(* CODESYS project XBoxControllerUtilities.library
   Author: John Helfrich
   Placeholder: XBoxControllerUtilities
   Title: XBoxControllerUtilities
   Version: 1.0
   Company: Beckhoff Community

Project tree, tasks and I/O mapping:
  libraries: Tc2_MC2, * (Beckhoff Automation GmbH); Tc2_Standard, * (Beckhoff Automation GmbH); Tc2_System, * (Beckhoff Automation GmbH); Tc3_Module, * (Beckhoff Automation GmbH)
  DUTs/
    LowerLevel/
      data type ST_XBox_Controller_Buttons_Bits
      data type ST_XBox_Controller_State_Bits2
    XBox NC/
      data type ST_XBox_Button_NC_Options
      data type ST_XBox_Dual_Directional_Joystick_NC_Options
      data type ST_XBox_Single_Directional_Joystick_NC_Options
      data type ST_XBox_Trigger_NC_Options
    data type E_XBox_Controller_Battery_Levels
    data type E_XBox_Controller_Battery_Types
    data type ST_XBox_Class_Command_Status
    data type ST_XBox_Controller_ADS_Inputs
    data type ST_XBox_Controller_Buttons
    data type ST_XBox_Controller_DPad
    data type ST_XBox_Controller_Joystick
    data type ST_XBox_Controller_Rumble
    data type ST_XBox_Controller_Status
  FBs/
    Base Gamepad/
      function block FB_XBox_Controller [ST]: Cycle, FB_init, P_Buttons, P_Left_Joystick, P_Left_Trigger, P_Right_Joystick, P_Right_Trigger, P_SetRumble, P_Status, SetRumble
    NC/
      Buttons/
        function block FB_XBox_Dual_Button_NC [ST]: FB_init, Jog
        function block FB_XBox_Single_Button_NC [ST]: FB_init, Jog
      Joysticks/
        function block FB_XBox_Dual_Directional_Joystick_NC [ST]: FB_init, Jog
        function block FB_XBox_Single_Directional_Joystick_NC [ST]: FB_init, Jog
      Triggers/
        function block FB_XBox_Dual_Trigger_NC [ST]: FB_init, Jog
        function block FB_XBox_Single_Trigger_NC [ST]: FB_init, Jog
  Project Information/
    function F_GetCompany [ST]
    function F_GetTitle [ST]
    function F_GetVersion [ST]
  Version/
    global variables Global_Version
*)

// DUTs/LowerLevel/ST_XBox_Controller_Buttons_Bits
TYPE ST_XBox_Controller_Buttons_Bits :
STRUCT
	xDPAD_UP  			: BIT;
    xDPAD_DOWN  		: BIT;
    xDPAD_LEFT  		: BIT;
    xDPAD_RIGHT  		: BIT;
    xSTART  			: BIT;
    xBACK  				: BIT;
    xLEFT_THUMB  		: BIT;
    xRIGHT_THUMB  		: BIT;   
	xLEFT_SHOULDER  	: BIT;
    xRIGHT_SHOULDER  	: BIT;
	{attribute 'hide'}
	xFiller1 			: BIT;
	{attribute 'hide'}
	xFiller2			: BIT;
	xA  				: BIT;
	xB  				: BIT;
	xX  				: BIT;
	xY  				: BIT;
END_STRUCT
END_TYPE

// DUTs/LowerLevel/ST_XBox_Controller_State_Bits2
TYPE ST_XBox_Controller_State_Bits2 :
STRUCT
	xConnected  				: BIT;
	xBattery_Type_Disconnected	: BIT;
	xBattery_Type_Wired			: BIT;
	xBattery_Type_Alkaline		: BIT;
	xBattery_Type_NIMH			: BIT;
	xBattery_Type_Unknown		: BIT;
	xBattery_Level_Empty		: BIT;
	xBattery_Level_Low			: BIT;
	xBattery_Level_Medium		: BIT;
	xBattery_Level_Full			: BIT;
	
	{attribute 'hide'}
	xFiller10					: BIT;
	{attribute 'hide'}
	xFiller11					: BIT;
	{attribute 'hide'}
	xFiller12					: BIT;
	{attribute 'hide'}
	xFiller13					: BIT;
	{attribute 'hide'}
	xFiller14					: BIT;
	{attribute 'hide'}
	xFiller15					: BIT;
END_STRUCT
END_TYPE

// DUTs/XBox NC/ST_XBox_Button_NC_Options
TYPE ST_XBox_Button_NC_Options :
STRUCT
	// Inverts the direction of the axis
	bInverted : BOOL := FALSE;
	// Maximum Feedrate
	fMaxOverride : LREAL := 100.0;
	// Ramped Feedrate - Increase the feedrate over time of button pressed
	bRampedOverride : BOOL := TRUE;
	// Ramp Step - How often to increase override as button is pressed
	tRampStepTime : TIME := T#100MS;
	// Ramp Step Factor - The % override to step at each time period
	iRampStepFactor : INT := 5;
END_STRUCT
END_TYPE

// DUTs/XBox NC/ST_XBox_Dual_Directional_Joystick_NC_Options
TYPE ST_XBox_Dual_Directional_Joystick_NC_Options :
STRUCT
	// Inverts the direction of the X axis
	bInverted_X : BOOL := FALSE;
	// Inverts the direction of the Y axis
	bInverted_Y : BOOL := FALSE;
	// Maximum Feedrate X Axis
	fMaxOverride_X : LREAL := 100.0;
	// Maximum Feedrate Y Axis
	fMaxOverride_Y : LREAL := 100.0;
END_STRUCT
END_TYPE

// DUTs/XBox NC/ST_XBox_Single_Directional_Joystick_NC_Options
TYPE ST_XBox_Single_Directional_Joystick_NC_Options :
STRUCT
	// Inverts the direction of the axis
	bInverted : BOOL := FALSE;
	// Maximum Feedrate
	fMaxOverride : LREAL := 100.0;
END_STRUCT
END_TYPE

// DUTs/XBox NC/ST_XBox_Trigger_NC_Options
TYPE ST_XBox_Trigger_NC_Options :
STRUCT
	// Inverts the direction of the axis
	bInverted : BOOL := FALSE;
	// Maximum Feedrate
	fMaxOverride : LREAL := 100.0;
END_STRUCT
END_TYPE

// DUTs/E_XBox_Controller_Battery_Levels
{attribute 'qualified_only'}
{attribute 'strict'}
TYPE E_XBox_Controller_Battery_Levels :
(
	// Battery is Empty or Unknown
	Empty := 0,
	// Battery is at low level
	Low := 1,
	// Battery is at medium level
	Medium := 2,
	// Battery is at full level
	Full := 3
);
END_TYPE

// DUTs/E_XBox_Controller_Battery_Types
{attribute 'qualified_only'}
{attribute 'strict'}
TYPE E_XBox_Controller_Battery_Types :
(
	// Battery is disconnected
	Disconnected := 0,
	// Battery is wired
	Wired := 1,
	// Battery is alkaline
	Alkaline := 2,
	// Battery is nickel-metal hydride
	NIMH := 3,
	// Battery is unknown
	Unknown := 4
);
END_TYPE

// DUTs/ST_XBox_Class_Command_Status
TYPE ST_XBox_Class_Command_Status :
STRUCT
	// Command has been completed
	bDone 	: BOOL;
	// Command is busy
	bBusy 	: BOOL;
	// Command has an error
	bError 	: BOOL;
END_STRUCT
END_TYPE

// DUTs/ST_XBox_Controller_ADS_Inputs
TYPE ST_XBox_Controller_ADS_Inputs :
STRUCT
	// Controller Number
	iControllerNumber	: INT;
	// Struct of Left Joystick values
	stLeft_Joystick 	: ST_XBox_Controller_Joystick;
	// Struct of Right Joystick values
	stRight_Joystick 	: ST_XBox_Controller_Joystick;
	// Left Trigger value
	fLeft_Trigger 		: REAL;
	// Right Trigger value
	fRight_Trigger 		: REAL;
	// Struct of individual raw button bits read from the controller
	bButtons 			: ST_XBox_Controller_Buttons_Bits;
	// Struct of individual raw status bits read from the controller
	bStatus				: ST_XBox_Controller_State_Bits2;
END_STRUCT
END_TYPE

// DUTs/ST_XBox_Controller_Buttons
TYPE ST_XBox_Controller_Buttons :
STRUCT
	// Directional Pad Struct
	DPad				: ST_XBox_Controller_DPad;
	// Start Button
    bStart  			: BOOL;
	// Back Button
    bBack  				: BOOL;
	// Pressing in the Left Thumbstick
    bLeft_Thumbstick  	: BOOL;
	// Pressing in the Right Thumbstick
    bRight_Thumbstick  	: BOOL;
	// Left Shoulder Button  
	bLeft_Shoulder  	: BOOL;
	// Right Shoulder Button
    bRight_Shoulder  	: BOOL;
	// Button A
	bA_Button  			: BOOL;
	// Button B
	bB_Button  			: BOOL;
	// Button X
	bX_Button  			: BOOL;
	// Button Y
	bY_Button  			: BOOL;
END_STRUCT
END_TYPE

// DUTs/ST_XBox_Controller_DPad
TYPE ST_XBox_Controller_DPad :
STRUCT
	// Up Button on DPad
	bUp  		: BOOL;
	// Down Button on DPad
    bDown  		: BOOL;
	// Left Button on DPad
    bLeft  		: BOOL;
	// Right Button on DPad
    bRight  	: BOOL;
END_STRUCT
END_TYPE

// DUTs/ST_XBox_Controller_Joystick
TYPE ST_XBox_Controller_Joystick :
STRUCT
	// Joystick's X Value (-100...100%)
	fX : REAL;
	// Joystick's Y Value (-100...100%)
	fY : REAL;
END_STRUCT
END_TYPE

// DUTs/ST_XBox_Controller_Rumble
TYPE ST_XBox_Controller_Rumble :
STRUCT
	// Rumble of left motor (0..100%)
	fLeftMotor 	: REAL;
	// Rumble of right motor (0..100%)
	fRightMotor : REAL;
END_STRUCT
END_TYPE

// DUTs/ST_XBox_Controller_Status
TYPE ST_XBox_Controller_Status :
STRUCT
	// Controller's ID
	iControllerNumber  	: INT;
	// Controller is connected to the PC
	bConnected  		: BOOL;
	// Controller is disconnected from the PC
	bDisconnected  		: BOOL;
	// Battery Type
	Battery_Type 		: E_XBox_Controller_Battery_Types;
	// Battery Level
	Battery_Level 		: E_XBox_Controller_Battery_Levels;
END_STRUCT
END_TYPE

// Version/Global_Version
{attribute 'TcGenerated'}
{attribute 'no-analysis'}
{attribute 'linkalways'}
// This function has been automatically generated from the project information.
VAR_GLOBAL CONSTANT
	{attribute 'const_non_replaced'}
	stLibVersion_XBoxControllerUtilities : ST_LibVersion := (iMajor := 1, iMinor := 0, iBuild := 0, iRevision := 0, nFlags := 1, sVersion := '1.0');
END_VAR

// FBs/Base Gamepad/FB_XBox_Controller
FUNCTION_BLOCK FB_XBox_Controller
VAR
	{attribute 'hide'}
	_AmsNetId : T_AMSNETID;
	{attribute 'hide'}
	_WriteServerData : ADSWRITE;
	{attribute 'hide'}
	_ReadServerData : ADSREAD;
	// RAW ADS Inputs for debug (Use properties to access items)
	stXBoxControllerInputs : ST_XBox_Controller_ADS_Inputs;
	{attribute 'hide'}
	_stRumble : ST_XBox_Controller_Rumble;
	{attribute 'hide'}
	_IDXGRP : UDINT;
	{attribute 'hide'}
	_rumbleCommand 			: ST_XBox_Class_Command_Status;
	{attribute 'hide'}
	_stControllerButtons 	: ST_XBox_Controller_Buttons;
	{attribute 'hide'}
	_stControllerStatus		: ST_XBox_Controller_Status;
	{attribute 'hide'}
	_stLeftJoystick 		: ST_XBox_Controller_Joystick;
	{attribute 'hide'}
	_stRightJoystick 		: ST_XBox_Controller_Joystick;
	{attribute 'hide'}
	_fLeftTrigger 			: REAL;
	{attribute 'hide'}
	_fRightTrigger 			: REAL;
	{attribute 'hide'}
	_bSetRumbleEvent 		: BOOL; // Internal indication of an ADS write event
	{attribute 'hide'}
	_bSetRumbleEventLogged	: BOOL; // Check if the Set Rumble event is being called too many times	
END_VAR

// This method is called cyclically to update the controller inputs
METHOD Cycle : BOOL
// Read the current inputs
THIS^._ReadServerData(
	NETID:= THIS^._AmsNetId, 
	PORT:= 25733, 
	IDXGRP:= THIS^._IDXGRP, 
	IDXOFFS:= 0, 
	LEN:= SIZEOF(THIS^.stXBoxControllerInputs), 
	DESTADDR:= ADR(THIS^.stXBoxControllerInputs), 
	READ:= TRUE, 
	TMOUT:= T#5S,
	ERR=>);
	
// If there is an error in reading from the server, shut all inputs off
IF THIS^._ReadServerData.ERR THEN
	memset(ADR(THIS^.stXBoxControllerInputs), 0, SIZEOF(THIS^.stXBoxControllerInputs));
END_IF

// Stop read command
THIS^._ReadServerData(
	NETID:= THIS^._AmsNetId, 
	PORT:= 25733, 
	IDXGRP:= THIS^._IDXGRP, 
	IDXOFFS:= 0, 
	LEN:= SIZEOF(THIS^.stXBoxControllerInputs), 
	DESTADDR:= ADR(THIS^.stXBoxControllerInputs), 
	READ:= FALSE, 
	TMOUT:= T#5S,
	ERR=>);
	

// Handle any write requests for the rumble
// Write the new values
THIS^._WriteServerData(
	NETID:= THIS^._AmsNetId, 
	PORT:= 25733, 
	IDXGRP:= THIS^._IDXGRP, 
	IDXOFFS:= 16, 
	LEN:= SIZEOF(THIS^._stRumble), 
	SRCADDR:= ADR(THIS^._stRumble), 
	WRITE:= THIS^._bSetRumbleEvent, 
	TMOUT:= T#5S);
	
// Update the status of the current command if active
IF 	THIS^._bSetRumbleEvent THEN
	THIS^.P_SetRumble.bBusy := THIS^._WriteServerData.BUSY;
	THIS^.P_SetRumble.bError := THIS^._WriteServerData.ERR;
END_IF

// Check if it's done writing
IF THIS^._bSetRumbleEvent AND NOT THIS^._WriteServerData.BUSY THEN
	IF NOT THIS^._WriteServerData.ERR THEN
		THIS^.P_SetRumble.bDone := TRUE;
	END_IF
	// Turn off the write request
	THIS^._WriteServerData(
		NETID:= THIS^._AmsNetId, 
		PORT:= 25733, 
		IDXGRP:= THIS^._IDXGRP, 
		IDXOFFS:= 16, 
		LEN:= SIZEOF(THIS^._stRumble), 
		SRCADDR:= ADR(THIS^._stRumble), 
		WRITE:= FALSE, 
		TMOUT:= T#5S);
		
	THIS^._bSetRumbleEvent := FALSE;
END_IF
END_METHOD

METHOD FB_init : BOOL
VAR_INPUT
	bInitRetains : BOOL; // if TRUE, the retain variables are initialized (warm start / cold start)
	bInCopyCode : BOOL;  // if TRUE, the instance afterwards gets moved into the copy code (online change)
	NetID 				: T_AMSNETID := ''; // AMS Net ID of the XBox Service Provider
	iControllerNumber 	: UINT(1..4) := 1; // The controller number for the controller you'd like to use
END_VAR
THIS^._AmsNetId := NetID;
THIS^._IDXGRP := iControllerNumber * 16#10000;
END_METHOD

// Structure of the different active buttons
PROPERTY P_Buttons : REFERENCE TO ST_XBox_Controller_Buttons
GET
IF THIS^.stXBoxControllerInputs.bStatus.xConnected THEN	
	THIS^._stControllerButtons.DPad.bUp				:= THIS^.stXBoxControllerInputs.bButtons.xDPAD_UP;
	THIS^._stControllerButtons.DPad.bDown			:= THIS^.stXBoxControllerInputs.bButtons.xDPAD_DOWN;
	THIS^._stControllerButtons.DPad.bLeft			:= THIS^.stXBoxControllerInputs.bButtons.xDPAD_LEFT;
	THIS^._stControllerButtons.DPad.bRight			:= THIS^.stXBoxControllerInputs.bButtons.xDPAD_RIGHT;
	THIS^._stControllerButtons.bStart  				:= THIS^.stXBoxControllerInputs.bButtons.xSTART;
	THIS^._stControllerButtons.bBack  				:= THIS^.stXBoxControllerInputs.bButtons.xBACK;
	THIS^._stControllerButtons.bLeft_Thumbstick  	:= THIS^.stXBoxControllerInputs.bButtons.xLEFT_THUMB;
	THIS^._stControllerButtons.bRight_Thumbstick 	:= THIS^.stXBoxControllerInputs.bButtons.xRIGHT_THUMB;
	THIS^._stControllerButtons.bLeft_Shoulder  		:= THIS^.stXBoxControllerInputs.bButtons.xLEFT_SHOULDER;
	THIS^._stControllerButtons.bRight_Shoulder  	:= THIS^.stXBoxControllerInputs.bButtons.xRIGHT_SHOULDER;
	THIS^._stControllerButtons.bA_Button  			:= THIS^.stXBoxControllerInputs.bButtons.xA;
	THIS^._stControllerButtons.bB_Button  			:= THIS^.stXBoxControllerInputs.bButtons.xB;
	THIS^._stControllerButtons.bX_Button  			:= THIS^.stXBoxControllerInputs.bButtons.xX;
	THIS^._stControllerButtons.bY_Button  			:= THIS^.stXBoxControllerInputs.bButtons.xY;
ELSE
	THIS^._stControllerButtons.DPad.bUp				:= FALSE;
	THIS^._stControllerButtons.DPad.bDown			:= FALSE;
	THIS^._stControllerButtons.DPad.bLeft			:= FALSE;
	THIS^._stControllerButtons.DPad.bRight			:= FALSE;
	THIS^._stControllerButtons.bStart  				:= FALSE;
	THIS^._stControllerButtons.bBack  				:= FALSE;
	THIS^._stControllerButtons.bLeft_Thumbstick  	:= FALSE;
	THIS^._stControllerButtons.bRight_Thumbstick 	:= FALSE;
	THIS^._stControllerButtons.bLeft_Shoulder  		:= FALSE;
	THIS^._stControllerButtons.bRight_Shoulder  	:= FALSE;
	THIS^._stControllerButtons.bA_Button  			:= FALSE;
	THIS^._stControllerButtons.bB_Button  			:= FALSE;
	THIS^._stControllerButtons.bX_Button  			:= FALSE;
	THIS^._stControllerButtons.bY_Button  			:= FALSE;
END_IF
P_Buttons REF= THIS^._stControllerButtons;
END_GET
END_PROPERTY

// Returns a structure of data for the XY Joystick values
PROPERTY P_Left_Joystick : REFERENCE TO ST_XBox_Controller_Joystick
GET
IF THIS^.stXBoxControllerInputs.bStatus.xConnected THEN	
	THIS^._stLeftJoystick.fX := THIS^.stXBoxControllerInputs.stLeft_Joystick.fX;
	THIS^._stLeftJoystick.fY := THIS^.stXBoxControllerInputs.stLeft_Joystick.fY;
ELSE
	THIS^._stLeftJoystick.fX := 0;
	THIS^._stLeftJoystick.fY := 0;
END_IF
P_Left_Joystick REF= THIS^._stLeftJoystick;
END_GET
END_PROPERTY

// Left trigger value
PROPERTY P_Left_Trigger : REFERENCE TO REAL
GET
IF THIS^.stXBoxControllerInputs.bStatus.xConnected THEN	
	THIS^._fLeftTrigger := THIS^.stXBoxControllerInputs.fLeft_Trigger;
ELSE
	THIS^._fLeftTrigger := 0;
END_IF
P_Left_Trigger REF= THIS^._fLeftTrigger;
END_GET
END_PROPERTY

// Returns a structure of data for the XY Joystick values
PROPERTY P_Right_Joystick : REFERENCE TO ST_XBox_Controller_Joystick
GET
IF THIS^.stXBoxControllerInputs.bStatus.xConnected THEN	
	THIS^._stRightJoystick.fX := THIS^.stXBoxControllerInputs.stRight_Joystick.fX;
	THIS^._stRightJoystick.fY := THIS^.stXBoxControllerInputs.stRight_Joystick.fY;
ELSE
	THIS^._stRightJoystick.fX := 0;
	THIS^._stRightJoystick.fY := 0;
END_IF
P_Right_Joystick REF= THIS^._stRightJoystick;
END_GET
END_PROPERTY

// Right trigger value
PROPERTY P_Right_Trigger : REFERENCE TO REAL
GET
IF THIS^.stXBoxControllerInputs.bStatus.xConnected THEN	
	THIS^._fRightTrigger := THIS^.stXBoxControllerInputs.fRight_Trigger;
ELSE
	THIS^._fRightTrigger := 0;
END_IF
P_Right_Trigger REF= THIS^._fRightTrigger;
END_GET
END_PROPERTY

// Status of the SetRumble method
PROPERTY P_SetRumble : REFERENCE TO ST_XBox_Class_Command_Status
GET
P_SetRumble REF= THIS^._rumbleCommand;
END_GET
END_PROPERTY

// Structure of the controller capabilites and status
PROPERTY P_Status : REFERENCE TO ST_XBox_Controller_Status
GET
IF THIS^.stXBoxControllerInputs.bStatus.xConnected THEN	
	THIS^._stControllerStatus.bConnected 		:= TRUE;
	THIS^._stControllerStatus.bDisconnected 	:= FALSE;
	THIS^._stControllerStatus.iControllerNumber := THIS^.stXBoxControllerInputs.iControllerNumber;
ELSE
	THIS^._stControllerStatus.bConnected 		:= FALSE;
	THIS^._stControllerStatus.bDisconnected 	:= TRUE;
	THIS^._stControllerStatus.iControllerNumber := 0;
END_IF

IF THIS^.stXBoxControllerInputs.bStatus.xBattery_Type_Disconnected THEN
	THIS^._stControllerStatus.Battery_Type := E_XBox_Controller_Battery_Types.Disconnected;
END_IF

IF THIS^.stXBoxControllerInputs.bStatus.xBattery_Type_Wired THEN
	THIS^._stControllerStatus.Battery_Type := E_XBox_Controller_Battery_Types.Wired;
END_IF

IF THIS^.stXBoxControllerInputs.bStatus.xBattery_Type_Alkaline THEN
	THIS^._stControllerStatus.Battery_Type := E_XBox_Controller_Battery_Types.Alkaline;
END_IF

IF THIS^.stXBoxControllerInputs.bStatus.xBattery_Type_NIMH THEN
	THIS^._stControllerStatus.Battery_Type := E_XBox_Controller_Battery_Types.NIMH;
END_IF

IF THIS^.stXBoxControllerInputs.bStatus.xBattery_Type_Unknown THEN
	THIS^._stControllerStatus.Battery_Type := E_XBox_Controller_Battery_Types.Unknown;
END_IF

IF THIS^.stXBoxControllerInputs.bStatus.xBattery_Level_Empty THEN
	THIS^._stControllerStatus.Battery_Level := E_XBox_Controller_Battery_Levels.Empty;
END_IF

IF THIS^.stXBoxControllerInputs.bStatus.xBattery_Level_Low THEN
	THIS^._stControllerStatus.Battery_Level := E_XBox_Controller_Battery_Levels.Low;
END_IF

IF THIS^.stXBoxControllerInputs.bStatus.xBattery_Level_Medium THEN
	THIS^._stControllerStatus.Battery_Level := E_XBox_Controller_Battery_Levels.Medium;
END_IF

IF THIS^.stXBoxControllerInputs.bStatus.xBattery_Level_Full THEN
	THIS^._stControllerStatus.Battery_Level := E_XBox_Controller_Battery_Levels.Full;
END_IF


P_Status REF= THIS^._stControllerStatus;
END_GET
END_PROPERTY

// Sets the rumble for the controller
METHOD SetRumble : BOOL
VAR_INPUT
	// Left motor speed (0..100%)
	fLeftMotor : REAL;
	// Right motor speed (0..100%)
	fRightMotor : REAL;
END_VAR
// When the method is called, check if a write is in progress
IF THIS^._bSetRumbleEvent THEN
	// ADS you are doing that too much
	IF NOT THIS^._bSetRumbleEventLogged THEN
		ADSLOGSTR( msgCtrlMask := ADSLOG_MSGTYPE_WARN, msgFmtStr := 'PLC Msg.: Command being called too often, wait for done bit: %s', strArg := 'SetRumble()');
		THIS^._bSetRumbleEventLogged := TRUE;
	END_IF	
ELSE
	// Check if the value is within range
	IF fLeftMotor > 100 THEN
		THIS^._stRumble.fLeftMotor := 100.0;
	ELSIF fLeftMotor < 0 THEN
		THIS^._stRumble.fLeftMotor := 0.0;
	ELSE
		THIS^._stRumble.fLeftMotor := fLeftMotor;
	END_IF
	
	// Check if the value is within range
	IF fRightMotor > 100 THEN
		THIS^._stRumble.fRightMotor := 100.0;
	ELSIF fRightMotor < 0 THEN
		THIS^._stRumble.fRightMotor := 0.0;
	ELSE
		THIS^._stRumble.fRightMotor := fRightMotor;
	END_IF
	
	//Reset all status for the command
	THIS^.P_SetRumble.bDone := FALSE;
	THIS^.P_SetRumble.bBusy := FALSE;
	THIS^.P_SetRumble.bError := FALSE;

	// Set the high bit on the write command
	THIS^._bSetRumbleEvent := TRUE;
END_IF

// If it's done, set the current even in progress to false
IF P_SetRumble.bDone THEN
	THIS^._bSetRumbleEvent := FALSE;
END_IF

// Event Received
SetRumble := THIS^._bSetRumbleEvent;
END_METHOD

END_FUNCTION_BLOCK

// FBs/NC/Buttons/FB_XBox_Dual_Button_NC
FUNCTION_BLOCK FB_XBox_Dual_Button_NC
VAR
	// Axis Control Blocks
	_Button_NC			: FB_XBox_Single_Button_NC;
	_rtJogEnable		: R_TRIG;
	_ftJogEnable		: F_TRIG;
	_fPrevOverride		: UDINT;
END_VAR

METHOD FB_init : BOOL
VAR_INPUT
	bInitRetains : BOOL; // if TRUE, the retain variables are initialized (warm start / cold start)
	bInCopyCode : BOOL;  // if TRUE, the instance afterwards gets moved into the copy code (online change)
END_VAR
END_METHOD

METHOD Jog : BOOL
VAR_INPUT
	bEnable				: BOOL;	
	bForward_Button		: BOOL;
	bBackwards_Button	: BOOL;
	Axis				: REFERENCE TO Axis_Ref;
	stOptions			: ST_XBox_Button_NC_Options;
END_VAR
VAR	
	stButtonOptions		: ST_XBox_Button_NC_Options;
	bButtonCommand		: BOOL;
END_VAR
// Rising edge trigger of the block enable
_rtJogEnable(CLK := bEnable);
// Falling edge trigger of the block enable
_ftJogEnable(CLK := bEnable);

IF __ISVALIDREF(Axis) THEN
	// Rising edge trigger of the block enable
	IF _rtJogEnable.Q THEN
		// Save the current override value before jogging
		THIS^._fPrevOverride := Axis.PlcToNc.Override;
	END_IF
	
	// Figure out what direction the axis should move
	IF bForward_Button AND bBackwards_Button THEN
		bButtonCommand := FALSE;
	ELSIF bForward_Button THEN
		bButtonCommand := bForward_Button;
		IF NOT stOptions.bInverted THEN
			stButtonOptions.bInverted := FALSE;
		ELSE
			stButtonOptions.bInverted := TRUE;
		END_IF
	ELSIF bBackwards_Button THEN
		bButtonCommand := bBackwards_Button;
		IF NOT stOptions.bInverted THEN
			stButtonOptions.bInverted := TRUE;
		ELSE
			stButtonOptions.bInverted := FALSE;
		END_IF
	ELSE
		bButtonCommand := FALSE;
	END_IF
	
	stButtonOptions.bRampedOverride := stOptions.bRampedOverride;
	stButtonOptions.fMaxOverride := stOptions.fMaxOverride;
	stButtonOptions.iRampStepFactor := stOptions.iRampStepFactor;
	stButtonOptions.tRampStepTime := stOptions.tRampStepTime;
	
	// Jog the axis
	_Button_NC.Jog(bEnable:= bEnable, bButton:= bButtonCommand, Axis:= Axis, stOptions:= stButtonOptions);
	
	// Falling edge trigger of the block enable
	IF _ftJogEnable.Q THEN
		// Restore the past override value before enable
		Axis.PlcToNc.Override := THIS^._fPrevOverride;
	END_IF
END_IF
END_METHOD

END_FUNCTION_BLOCK

// FBs/NC/Buttons/FB_XBox_Single_Button_NC
FUNCTION_BLOCK FB_XBox_Single_Button_NC
VAR
	_mcJog				: MC_Jog;
	_rtJogEnable		: R_TRIG;
	_ftJogEnable		: F_TRIG;
	_bJoggingActive		: BOOL;
	_fPrevOverride		: UDINT;
	_RampTimer			: TON;
	_fCurrentOverride   : LREAL;
END_VAR

METHOD FB_init : BOOL
VAR_INPUT
	bInitRetains : BOOL; // if TRUE, the retain variables are initialized (warm start / cold start)
	bInCopyCode : BOOL;  // if TRUE, the instance afterwards gets moved into the copy code (online change)
END_VAR
END_METHOD

METHOD Jog : BOOL
VAR_INPUT
	bEnable			: BOOL;	
	bButton			: BOOL;
	Axis			: REFERENCE TO Axis_Ref;
	stOptions		: ST_XBox_Button_NC_Options;
END_VAR
VAR
	bJogForward 	 : BOOL;
	bJogBackwards 	 : BOOL;
END_VAR
// Rising edge trigger of the block enable
_rtJogEnable(CLK := bEnable);
// Falling edge trigger of the block enable
_ftJogEnable(CLK := bEnable);

// Rising edge trigger of the block enable
IF _rtJogEnable.Q THEN
	// Save the current override value before jogging
	// Check the Axis reference is valid	
	IF __ISVALIDREF(Axis) THEN
		THIS^._fPrevOverride := Axis.PlcToNc.Override;
	END_IF
	// Enable the jog methods
	_bJoggingActive	:= TRUE;
END_IF

// Falling edge trigger of the block enable
IF _ftJogEnable.Q THEN
	// Restore the past override value before enable
	// Check the Axis reference is valid	
	IF __ISVALIDREF(Axis) THEN
		Axis.PlcToNc.Override := THIS^._fPrevOverride;
			// Cleanup any old Jog commands
		THIS^._mcJog(
					  Axis:= Axis, 
					  JogForward:= FALSE, 
					  JogBackwards:= FALSE, 
					  Mode:= E_JogMode.MC_JOGMODE_STANDARD_FAST);	
	END_IF
	// Disable calling to jog methods
	_bJoggingActive := FALSE;
END_IF

// Check the Joystick reference is valid
IF _bJoggingActive THEN
	// Check the Axis reference is valid	
	IF __ISVALIDREF(Axis) THEN
		// Speed Ramp Timer
		_RampTimer(IN:=stOptions.bRampedOverride AND NOT _RampTimer.Q, PT:= stOptions.tRampStepTime);
		
		// Check the direction the joystick is moving, or if in deadzone					 
		IF bButton = FALSE THEN
			bJogForward 	:= FALSE;
			bJogBackwards := FALSE;
			Axis.PlcToNc.Override := 0;
			_fCurrentOverride := 0;
		ELSE
			// Check for inversion
			IF NOT stOptions.bInverted THEN
				bJogForward 	:= TRUE;
				bJogBackwards 	:= FALSE;
			ELSE
				bJogForward 	:= FALSE;
				bJogBackwards 	:= TRUE;
			END_IF
			
			// Find the override speed

			IF _RampTimer.Q AND stOptions.bRampedOverride THEN
				_fCurrentOverride := _fCurrentOverride + stOptions.iRampStepFactor;		
			ELSIF NOT stOptions.bRampedOverride THEN
				_fCurrentOverride := stOptions.fMaxOverride;
			END_IF
			// Check range
			IF _fCurrentOverride > stOptions.fMaxOverride THEN
				_fCurrentOverride := stOptions.fMaxOverride;
			END_IF
			
			Axis.PlcToNc.Override := TO_UDINT(ABS(_fCurrentOverride) * 10000);
		END_IF
		
		// Main jog call for axis
		THIS^._mcJog(
					  Axis:= Axis, 
					  JogForward:= bJogForward, 
					  JogBackwards:= bJogBackwards, 
					  Mode:= E_JogMode.MC_JOGMODE_STANDARD_FAST);
	END_IF
END_IF
END_METHOD

END_FUNCTION_BLOCK

// FBs/NC/Joysticks/FB_XBox_Dual_Directional_Joystick_NC
FUNCTION_BLOCK FB_XBox_Dual_Directional_Joystick_NC
VAR
	// Axis Control Blocks
	_JoystickNC_X		: FB_XBox_Single_Directional_Joystick_NC;
	_JoystickNC_Y		: FB_XBox_Single_Directional_Joystick_NC;
END_VAR

METHOD FB_init : BOOL
VAR_INPUT
	bInitRetains : BOOL; // if TRUE, the retain variables are initialized (warm start / cold start)
	bInCopyCode : BOOL;  // if TRUE, the instance afterwards gets moved into the copy code (online change)
END_VAR
END_METHOD

METHOD Jog
VAR_INPUT
	bEnable			: BOOL;	
	stJoystick		: REFERENCE TO ST_XBox_Controller_Joystick;
	X_Axis			: REFERENCE TO Axis_Ref;
	Y_Axis			: REFERENCE TO Axis_Ref;
	stOptions		: ST_XBox_Dual_Directional_Joystick_NC_Options;
END_VAR
VAR	
	X_Axis_Options: ST_XBox_Single_Directional_Joystick_NC_Options;
	Y_Axis_Options: ST_XBox_Single_Directional_Joystick_NC_Options;
END_VAR
IF __ISVALIDREF(stJoystick) AND __ISVALIDREF(X_Axis) AND __ISVALIDREF(Y_Axis) THEN
	// Call the X-Axis Joystick
	X_Axis_Options.bInverted := stOptions.bInverted_X;
	X_Axis_Options.fMaxOverride := stOptions.fMaxOverride_X;
	_JoystickNC_X.Jog(bEnable:= bEnable, fJoystick:= stJoystick.fX, Axis:= X_Axis, stOptions:= X_Axis_Options);
	
	// Call the Y-Axis Joystick
	Y_Axis_Options.bInverted := stOptions.bInverted_Y;
	Y_Axis_Options.fMaxOverride := stOptions.fMaxOverride_Y;
	_JoystickNC_Y.Jog(bEnable:= bEnable, fJoystick:= stJoystick.fY, Axis:= Y_Axis, stOptions:= Y_Axis_Options);
END_IF
END_METHOD

END_FUNCTION_BLOCK

// FBs/NC/Joysticks/FB_XBox_Single_Directional_Joystick_NC
FUNCTION_BLOCK FB_XBox_Single_Directional_Joystick_NC
VAR
	_mcJog				: MC_Jog;
	_rtJogEnable		: R_TRIG;
	_ftJogEnable		: F_TRIG;
	_bJoggingActive		: BOOL;
	_fPrevOverride		: UDINT;
END_VAR

METHOD FB_init : BOOL
VAR_INPUT
	bInitRetains : BOOL; // if TRUE, the retain variables are initialized (warm start / cold start)
	bInCopyCode : BOOL;  // if TRUE, the instance afterwards gets moved into the copy code (online change)
END_VAR
END_METHOD

METHOD Jog
VAR_INPUT
	bEnable			: BOOL;	
	fJoystick		: LREAL;
	Axis			: REFERENCE TO Axis_Ref;
	stOptions		: ST_XBox_Single_Directional_Joystick_NC_Options;
END_VAR
VAR
	bJogForward 	: BOOL;
	bJogBackwards 	: BOOL;
END_VAR
// Rising edge trigger of the block enable
_rtJogEnable(CLK := bEnable);
// Falling edge trigger of the block enable
_ftJogEnable(CLK := bEnable);

// Rising edge trigger of the block enable
IF _rtJogEnable.Q THEN
	// Save the current override value before jogging
	// Check the Axis reference is valid	
	IF __ISVALIDREF(Axis) THEN
		THIS^._fPrevOverride := Axis.PlcToNc.Override;
	END_IF
	// Enable the jog methods
	_bJoggingActive	:= TRUE;
END_IF

// Falling edge trigger of the block enable
IF _ftJogEnable.Q THEN
	// Restore the past override value before enable
	// Check the Axis reference is valid	
	IF __ISVALIDREF(Axis) THEN
		Axis.PlcToNc.Override := THIS^._fPrevOverride;
			// Cleanup any old Jog commands
		THIS^._mcJog(
					  Axis:= Axis, 
					  JogForward:= FALSE, 
					  JogBackwards:= FALSE, 
					  Mode:= E_JogMode.MC_JOGMODE_STANDARD_FAST);	
	END_IF
	// Disable calling to jog methods
	_bJoggingActive := FALSE;
END_IF

// Check the Joystick reference is valid
IF _bJoggingActive THEN
	// Check the Axis reference is valid	
	IF __ISVALIDREF(Axis) THEN
		// Check the direction the joystick is moving, or if in deadzone					 
		IF fJoystick = 0 THEN
			bJogForward 	:= FALSE;
			bJogBackwards := FALSE;
			Axis.PlcToNc.Override := 0;
		ELSIF fJoystick < 0 THEN
			// Check for inversion
			IF NOT stOptions.bInverted THEN
				bJogForward 	:= FALSE;
				bJogBackwards := TRUE;
			ELSE
				bJogForward 	:= TRUE;
				bJogBackwards := FALSE;
			END_IF
			// Set the new override based on the directional pressure
			Axis.PlcToNc.Override := TO_UDINT(ABS(fJoystick * (stOptions.fMaxOverride/100)) * 10000);
		ELSIF fJoystick > 0 THEN
			// Check for inversion
			IF NOT stOptions.bInverted THEN
				bJogForward 	:= TRUE;
				bJogBackwards := FALSE;
			ELSE
				bJogForward 	:= FALSE;
				bJogBackwards := TRUE;
			END_IF
			// Set the new override based on the directional pressure
			Axis.PlcToNc.Override := TO_UDINT(ABS(fJoystick * (stOptions.fMaxOverride/100)) * 10000);
		END_IF
		// Main jog call for axis
		THIS^._mcJog(
					  Axis:= Axis, 
					  JogForward:= bJogForward, 
					  JogBackwards:= bJogBackwards, 
					  Mode:= E_JogMode.MC_JOGMODE_STANDARD_FAST);
	END_IF
END_IF
END_METHOD

END_FUNCTION_BLOCK

// FBs/NC/Triggers/FB_XBox_Dual_Trigger_NC
FUNCTION_BLOCK FB_XBox_Dual_Trigger_NC
VAR
	// Axis Control Blocks
	_Trigger_NC			: FB_XBox_Single_Trigger_NC;
	_rtJogEnable		: R_TRIG;
	_ftJogEnable		: F_TRIG;
	_fPrevOverride		: UDINT;
END_VAR

METHOD FB_init : BOOL
VAR_INPUT
	bInitRetains : BOOL; // if TRUE, the retain variables are initialized (warm start / cold start)
	bInCopyCode : BOOL;  // if TRUE, the instance afterwards gets moved into the copy code (online change)
END_VAR
END_METHOD

METHOD Jog
VAR_INPUT
	bEnable			: BOOL;	
	fLeft_Trigger	: LREAL;
	fRight_Trigger	: LREAL;
	Axis			: REFERENCE TO Axis_Ref;
	stOptions		: ST_XBox_Trigger_NC_Options;
END_VAR
VAR	
	stTrigOptions		: ST_XBox_Trigger_NC_Options;
	fTriggerCommand		: LREAL;
END_VAR
// Rising edge trigger of the block enable
_rtJogEnable(CLK := bEnable);
// Falling edge trigger of the block enable
_ftJogEnable(CLK := bEnable);

IF __ISVALIDREF(Axis) THEN
	// Rising edge trigger of the block enable
	IF _rtJogEnable.Q THEN
		// Save the current override value before jogging
		THIS^._fPrevOverride := Axis.PlcToNc.Override;
	END_IF
	
	// Figure out what direction the axis should move
	IF fLeft_Trigger > fRight_Trigger THEN
		fTriggerCommand := fLeft_Trigger;
		IF NOT stOptions.bInverted THEN
			stTrigOptions.bInverted := FALSE;
		ELSE
			stTrigOptions.bInverted := TRUE;
		END_IF
	ELSIF fRight_Trigger > fLeft_Trigger THEN
		fTriggerCommand := fRight_Trigger;
		IF NOT stOptions.bInverted THEN
			stTrigOptions.bInverted := TRUE;
		ELSE
			stTrigOptions.bInverted := FALSE;
		END_IF
	ELSE
		fTriggerCommand := 0;
	END_IF
	stTrigOptions.fMaxOverride := stOptions.fMaxOverride;
	// Jog the axis
	_Trigger_NC.Jog(bEnable:= bEnable, fTrigger:= fTriggerCommand, Axis:= Axis, stOptions:= stTrigOptions);
	
	
	// Falling edge trigger of the block enable
	IF _ftJogEnable.Q THEN
		// Restore the past override value before enable
		Axis.PlcToNc.Override := THIS^._fPrevOverride;
	END_IF
END_IF
END_METHOD

END_FUNCTION_BLOCK

// FBs/NC/Triggers/FB_XBox_Single_Trigger_NC
FUNCTION_BLOCK FB_XBox_Single_Trigger_NC
VAR
	_mcJog				: MC_Jog;
	_rtJogEnable		: R_TRIG;
	_ftJogEnable		: F_TRIG;
	_bJoggingActive		: BOOL;
	_fPrevOverride		: UDINT;
END_VAR

METHOD FB_init : BOOL
VAR_INPUT
	bInitRetains : BOOL; // if TRUE, the retain variables are initialized (warm start / cold start)
	bInCopyCode : BOOL;  // if TRUE, the instance afterwards gets moved into the copy code (online change)
END_VAR
END_METHOD

METHOD Jog
VAR_INPUT
	bEnable			: BOOL;	
	fTrigger		: LREAL;
	Axis			: REFERENCE TO Axis_Ref;
	stOptions		: ST_XBox_Trigger_NC_Options;
END_VAR
VAR
	bJogForward 	: BOOL;
	bJogBackwards 	: BOOL;
END_VAR
// Rising edge trigger of the block enable
_rtJogEnable(CLK := bEnable);
// Falling edge trigger of the block enable
_ftJogEnable(CLK := bEnable);

// Rising edge trigger of the block enable
IF _rtJogEnable.Q THEN
	// Save the current override value before jogging
	// Check the Axis reference is valid	
	IF __ISVALIDREF(Axis) THEN
		THIS^._fPrevOverride := Axis.PlcToNc.Override;
	END_IF
	// Enable the jog methods
	_bJoggingActive	:= TRUE;
END_IF

// Falling edge trigger of the block enable
IF _ftJogEnable.Q THEN
	// Restore the past override value before enable
	// Check the Axis reference is valid	
	IF __ISVALIDREF(Axis) THEN
		Axis.PlcToNc.Override := THIS^._fPrevOverride;
			// Cleanup any old Jog commands
		THIS^._mcJog(
					  Axis:= Axis, 
					  JogForward:= FALSE, 
					  JogBackwards:= FALSE, 
					  Mode:= E_JogMode.MC_JOGMODE_STANDARD_FAST);	
	END_IF
	// Disable calling to jog methods
	_bJoggingActive := FALSE;
END_IF

// Check the Joystick reference is valid
IF _bJoggingActive THEN
	// Check the Axis reference is valid	
	IF __ISVALIDREF(Axis) THEN
		// Check the direction the joystick is moving, or if in deadzone					 
		IF fTrigger = 0 THEN
			bJogForward 	:= FALSE;
			bJogBackwards := FALSE;
			Axis.PlcToNc.Override := 0;
		ELSE
			// Check for inversion
			IF NOT stOptions.bInverted THEN
				bJogForward 	:= TRUE;
				bJogBackwards := FALSE;
			ELSE
				bJogForward 	:= FALSE;
				bJogBackwards := TRUE;
			END_IF
			// Set the new override based on the directional pressure
			Axis.PlcToNc.Override := TO_UDINT(ABS(fTrigger  * (stOptions.fMaxOverride/100)) * 10000);
		END_IF
		
		// Main jog call for axis
		THIS^._mcJog(
					  Axis:= Axis, 
					  JogForward:= bJogForward, 
					  JogBackwards:= bJogBackwards, 
					  Mode:= E_JogMode.MC_JOGMODE_STANDARD_FAST);
	END_IF
END_IF
END_METHOD

END_FUNCTION_BLOCK

// Project Information/F_GetCompany
// This function has been automatically generated from the project information.
{attribute 'signature_flag' := '1073741824'}
{attribute 'TcGenerated'}
{attribute 'no-analysis'}
FUNCTION F_GetCompany : WSTRING
VAR_INPUT
	
END_VAR

F_GetCompany := "Beckhoff Community";

END_FUNCTION

// Project Information/F_GetTitle
// This function has been automatically generated from the project information.
{attribute 'signature_flag' := '1073741824'}
{attribute 'TcGenerated'}
{attribute 'no-analysis'}
FUNCTION F_GetTitle : WSTRING
VAR_INPUT
	
END_VAR

F_GetTitle := "XBoxControllerUtilities";

END_FUNCTION

// Project Information/F_GetVersion
// This function has been automatically generated from the project information.
{attribute 'signature_flag' := '1073741824'}
{attribute 'TcGenerated'}
{attribute 'no-analysis'}
FUNCTION F_GetVersion : ST_LibVersion
VAR_INPUT
	
END_VAR

F_GetVersion.iMajor := 1;
F_GetVersion.iMinor := 0;
F_GetVersion.iBuild := 0;
F_GetVersion.iRevision := 0;
F_GetVersion.sVersion := '1.0';
F_GetVersion.nFlags := 1;

END_FUNCTION
